// Mitsubishi GX Works2 project: 비트별로동작   PLC: Q02/Q02H

PROGRAM MAIN
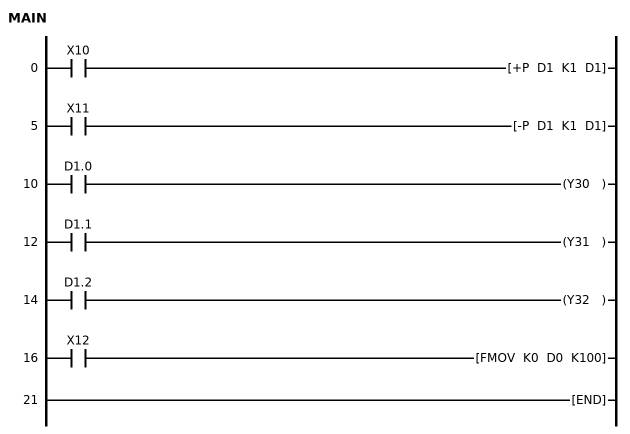
0     LD      X10
      +P      D1 K1 D1
5     LD      X11
      -P      D1 K1 D1
10    LD      D1.0
      OUT     Y30
12    LD      D1.1
      OUT     Y31
14    LD      D1.2
      OUT     Y32
16    LD      X12
      FMOV    K0 D0 K100
21    END
END_PROGRAM
